// TIA Portal project "Practica_7" (V13)

(* hardware
DEVICE "S7-1200 station_1"  S7-1200 Station
   slot 0: "Rack_0"  Rack  V1.0
   slot 1: "PLC_1"  Unspecific CPU 1200  6ES7 2XX-XXXXX-XXXX  V4.1
*)

// ===== PLC "PLC_1"  Unspecific CPU 1200 =====

VAR_GLOBAL   // PLC tag table "Default tag table"
   "PM(1)" AT %I0.0 : Bool;
   "PP(1)" AT %I0.1 : Bool;
   "M" AT %Q0.0 : Bool;
   "APAGADO" AT %M0.1 : Bool;
   "CNT" AT %M0.2 : Bool;
   "ENCENDIDO" AT %M0.0 : Bool;
   "PM" AT %M1.0 : Bool;
   "PP" AT %M1.1 : Bool;
   "IL" AT %Q0.1 : Bool;
   "DP" AT %I0.2 : Bool;
   "CU" AT %M0.3 : Bool;
END_VAR

// folder: System blocks/Program resources

DATA_BLOCK "CNT_UP"   // DB1
{ S7_Optimized_Access := 'FALSE' }
AUTHOR : Simatic
FAMILY : IEC
NAME : CNTR
VERSION : 1.0
// stored: InstanceOfName ?
"?"
BEGIN
END_DATA_BLOCK

// folder: (top level)

ORGANIZATION_BLOCK "Main"   // OB1, LAD, ProgramCycle
TITLE = "Main Program Sweep (Cycle)"
{ S7_Optimized_Access := 'FALSE' }
VERSION : 0.1
BEGIN

REGION Network 1
   // Marcha / Parada con autoretención
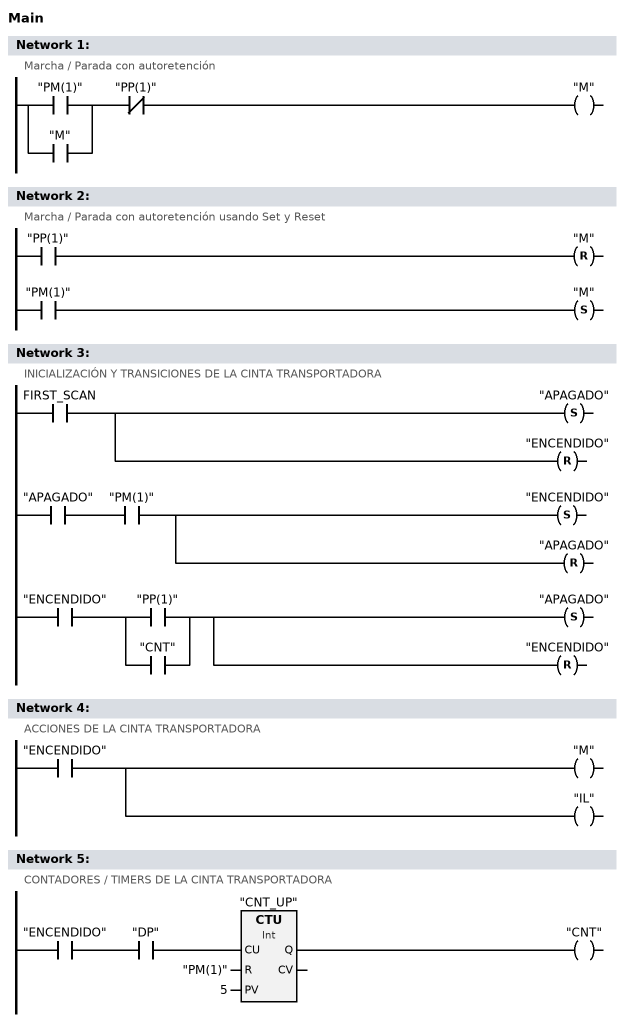
   RUNG wire#powerrail
      Contact( "PM(1)" )
      wire#w1
      I_Contact( "PP(1)" )
      Coil( "M" )
   END_RUNG
   RUNG wire#powerrail
      Contact( "M" )
   END_RUNG wire#w1
   // the same network as SCL:
   "M" := ("PM(1)" OR "M") AND NOT "PP(1)";
END_REGION

REGION Network 2
   // Marcha / Parada con autoretención usando Set y Reset
   RUNG wire#powerrail
      Contact( "PP(1)" )
      R_Coil( "M" )
   END_RUNG
   RUNG wire#powerrail
      Contact( "PM(1)" )
      S_Coil( "M" )
   END_RUNG
   // the same network as SCL:
   IF "PP(1)" THEN "M" := FALSE; END_IF;
   IF "PM(1)" THEN "M" := TRUE; END_IF;
END_REGION

REGION Network 3
   // INICIALIZACIÓN Y TRANSICIONES DE LA CINTA TRANSPORTADORA
   RUNG wire#powerrail
      Contact( FIRST_SCAN )
      wire#w1
      S_Coil( "APAGADO" )
   END_RUNG
   RUNG wire#w1
      R_Coil( "ENCENDIDO" )
   END_RUNG
   RUNG wire#powerrail
      Contact( "APAGADO" )
      Contact( "PM(1)" )
      wire#w2
      S_Coil( "ENCENDIDO" )
   END_RUNG
   RUNG wire#w2
      R_Coil( "APAGADO" )
   END_RUNG
   RUNG wire#powerrail
      Contact( "ENCENDIDO" )
      wire#w3
      Contact( "PP(1)" )
      wire#w4
      S_Coil( "APAGADO" )
   END_RUNG
   RUNG wire#w3
      Contact( "CNT" )
   END_RUNG wire#w4
   RUNG wire#w4
      R_Coil( "ENCENDIDO" )
   END_RUNG
   // the same network as SCL:
   IF FIRST_SCAN THEN
       "APAGADO" := TRUE;
       "ENCENDIDO" := FALSE;
   END_IF;
   IF "APAGADO" AND "PM(1)" THEN
       "ENCENDIDO" := TRUE;
       "APAGADO" := FALSE;
   END_IF;
   IF "ENCENDIDO" AND ("PP(1)" OR "CNT") THEN
       "APAGADO" := TRUE;
       "ENCENDIDO" := FALSE;
   END_IF;
END_REGION

REGION Network 4
   // ACCIONES DE LA CINTA TRANSPORTADORA
   RUNG wire#powerrail
      Contact( "ENCENDIDO" )
      wire#w1
      Coil( "M" )
   END_RUNG
   RUNG wire#w1
      Coil( "IL" )
   END_RUNG
   // the same network as SCL:
   "M" := "ENCENDIDO";
   "IL" := "ENCENDIDO";
END_REGION

REGION Network 5
   // CONTADORES / TIMERS DE LA CINTA TRANSPORTADORA
   "CNT_UP".CTU(CU := "ENCENDIDO" AND "DP", R := "PM(1)", PV := 5);
   "CNT" := "CNT_UP".Q;
END_REGION
END_ORGANIZATION_BLOCK